TYPE ST_BaseRecipeListRow :
STRUCT
	wsText			: WSTRING;
	iNumber			: INT;
	refRecipe		: REFERENCE TO ST_BaseRecipe;
END_STRUCT
END_TYPE

(* stored: Version 1.1.0.1
   DUT ST_BaseRecipeListRow: Id {25f5150b-f32b-0a24-1a7a-4eedc0019634} *)
